FUNCTION_BLOCK NORMALIZE
  {SET_ATTRIBUTE(OpcUa, SERVICE)}
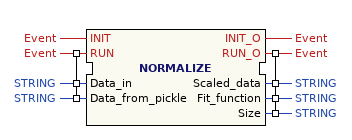
  EVENT_INPUT
    INIT;
    RUN WITH Data_in, Data_from_pickle; {SET_ATTRIBUTE(OpcUa, Method)}
  END_EVENT
  EVENT_OUTPUT
    INIT_O;
    RUN_O WITH Scaled_data, Fit_function, Size;
  END_EVENT
  VAR_INPUT
    Data_in : STRING; {SET_ATTRIBUTE(OpcUa, Variable.RUN)}
    Data_from_pickle : STRING; {SET_ATTRIBUTE(OpcUa, Variable.RUN)}
  END_VAR
  VAR_OUTPUT
    Scaled_data : STRING; {SET_ATTRIBUTE(OpcUa, Variable.RUN)}
    Fit_function : STRING; {SET_ATTRIBUTE(OpcUa, Variable.RUN)}
    Size : STRING; {SET_ATTRIBUTE(OpcUa, Variable.RUN)}
  END_VAR
END_FUNCTION_BLOCK
